FUNCTION_BLOCK SPLIT_AL_INTO_AX (* this Function splits the 64 AX (BOOL) adapters from a AL (LWORD) *)
  (* Standard: 61499-2; Description: Copyright (c) 2026 Meisterschulen am Ostbahnhof SPDX-License-Identifier: EPL-2.0 *)
  (* Version 1.0, 2026-05-16, Franz Höpfinger, Meisterschulen am Ostbahnhof, initial API and implementation and/or initial documentation *)
  PACKAGE adapter::splitting;
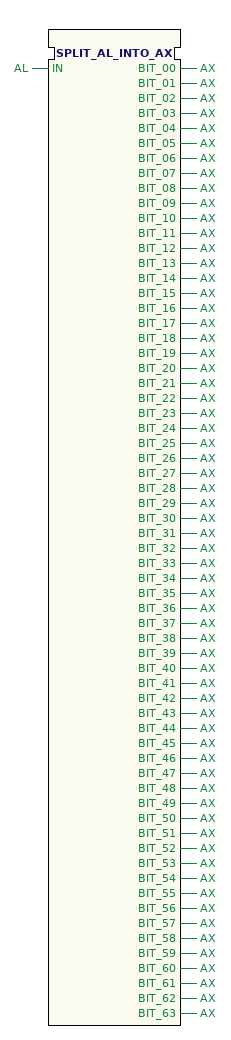
  SOCKETS
    IN : adapter::types::unidirectional::AL; (* LWORD Input *)
  END_SOCKETS
  PLUGS
    BIT_00 : adapter::types::unidirectional::AX; (* Bool Bit 0 *)
    BIT_01 : adapter::types::unidirectional::AX; (* Bool Bit 1 *)
    BIT_02 : adapter::types::unidirectional::AX; (* Bool Bit 2 *)
    BIT_03 : adapter::types::unidirectional::AX; (* Bool Bit 3 *)
    BIT_04 : adapter::types::unidirectional::AX; (* Bool Bit 4 *)
    BIT_05 : adapter::types::unidirectional::AX; (* Bool Bit 5 *)
    BIT_06 : adapter::types::unidirectional::AX; (* Bool Bit 6 *)
    BIT_07 : adapter::types::unidirectional::AX; (* Bool Bit 7 *)
    BIT_08 : adapter::types::unidirectional::AX; (* Bool Bit 8 *)
    BIT_09 : adapter::types::unidirectional::AX; (* Bool Bit 9 *)
    BIT_10 : adapter::types::unidirectional::AX; (* Bool Bit 10 *)
    BIT_11 : adapter::types::unidirectional::AX; (* Bool Bit 11 *)
    BIT_12 : adapter::types::unidirectional::AX; (* Bool Bit 12 *)
    BIT_13 : adapter::types::unidirectional::AX; (* Bool Bit 13 *)
    BIT_14 : adapter::types::unidirectional::AX; (* Bool Bit 14 *)
    BIT_15 : adapter::types::unidirectional::AX; (* Bool Bit 15 *)
    BIT_16 : adapter::types::unidirectional::AX; (* Bool Bit 16 *)
    BIT_17 : adapter::types::unidirectional::AX; (* Bool Bit 17 *)
    BIT_18 : adapter::types::unidirectional::AX; (* Bool Bit 18 *)
    BIT_19 : adapter::types::unidirectional::AX; (* Bool Bit 19 *)
    BIT_20 : adapter::types::unidirectional::AX; (* Bool Bit 20 *)
    BIT_21 : adapter::types::unidirectional::AX; (* Bool Bit 21 *)
    BIT_22 : adapter::types::unidirectional::AX; (* Bool Bit 22 *)
    BIT_23 : adapter::types::unidirectional::AX; (* Bool Bit 23 *)
    BIT_24 : adapter::types::unidirectional::AX; (* Bool Bit 24 *)
    BIT_25 : adapter::types::unidirectional::AX; (* Bool Bit 25 *)
    BIT_26 : adapter::types::unidirectional::AX; (* Bool Bit 26 *)
    BIT_27 : adapter::types::unidirectional::AX; (* Bool Bit 27 *)
    BIT_28 : adapter::types::unidirectional::AX; (* Bool Bit 28 *)
    BIT_29 : adapter::types::unidirectional::AX; (* Bool Bit 29 *)
    BIT_30 : adapter::types::unidirectional::AX; (* Bool Bit 30 *)
    BIT_31 : adapter::types::unidirectional::AX; (* Bool Bit 31 *)
    BIT_32 : adapter::types::unidirectional::AX; (* Bool Bit 32 *)
    BIT_33 : adapter::types::unidirectional::AX; (* Bool Bit 33 *)
    BIT_34 : adapter::types::unidirectional::AX; (* Bool Bit 34 *)
    BIT_35 : adapter::types::unidirectional::AX; (* Bool Bit 35 *)
    BIT_36 : adapter::types::unidirectional::AX; (* Bool Bit 36 *)
    BIT_37 : adapter::types::unidirectional::AX; (* Bool Bit 37 *)
    BIT_38 : adapter::types::unidirectional::AX; (* Bool Bit 38 *)
    BIT_39 : adapter::types::unidirectional::AX; (* Bool Bit 39 *)
    BIT_40 : adapter::types::unidirectional::AX; (* Bool Bit 40 *)
    BIT_41 : adapter::types::unidirectional::AX; (* Bool Bit 41 *)
    BIT_42 : adapter::types::unidirectional::AX; (* Bool Bit 42 *)
    BIT_43 : adapter::types::unidirectional::AX; (* Bool Bit 43 *)
    BIT_44 : adapter::types::unidirectional::AX; (* Bool Bit 44 *)
    BIT_45 : adapter::types::unidirectional::AX; (* Bool Bit 45 *)
    BIT_46 : adapter::types::unidirectional::AX; (* Bool Bit 46 *)
    BIT_47 : adapter::types::unidirectional::AX; (* Bool Bit 47 *)
    BIT_48 : adapter::types::unidirectional::AX; (* Bool Bit 48 *)
    BIT_49 : adapter::types::unidirectional::AX; (* Bool Bit 49 *)
    BIT_50 : adapter::types::unidirectional::AX; (* Bool Bit 50 *)
    BIT_51 : adapter::types::unidirectional::AX; (* Bool Bit 51 *)
    BIT_52 : adapter::types::unidirectional::AX; (* Bool Bit 52 *)
    BIT_53 : adapter::types::unidirectional::AX; (* Bool Bit 53 *)
    BIT_54 : adapter::types::unidirectional::AX; (* Bool Bit 54 *)
    BIT_55 : adapter::types::unidirectional::AX; (* Bool Bit 55 *)
    BIT_56 : adapter::types::unidirectional::AX; (* Bool Bit 56 *)
    BIT_57 : adapter::types::unidirectional::AX; (* Bool Bit 57 *)
    BIT_58 : adapter::types::unidirectional::AX; (* Bool Bit 58 *)
    BIT_59 : adapter::types::unidirectional::AX; (* Bool Bit 59 *)
    BIT_60 : adapter::types::unidirectional::AX; (* Bool Bit 60 *)
    BIT_61 : adapter::types::unidirectional::AX; (* Bool Bit 61 *)
    BIT_62 : adapter::types::unidirectional::AX; (* Bool Bit 62 *)
    BIT_63 : adapter::types::unidirectional::AX; (* Bool Bit 63 *)
  END_PLUGS
  FBS
    E_D_FF_00 : iec61499::events::E_D_FF;
    E_D_FF_01 : iec61499::events::E_D_FF;
    E_D_FF_02 : iec61499::events::E_D_FF;
    E_D_FF_03 : iec61499::events::E_D_FF;
    E_D_FF_04 : iec61499::events::E_D_FF;
    E_D_FF_05 : iec61499::events::E_D_FF;
    E_D_FF_06 : iec61499::events::E_D_FF;
    E_D_FF_07 : iec61499::events::E_D_FF;
    E_D_FF_08 : iec61499::events::E_D_FF;
    E_D_FF_09 : iec61499::events::E_D_FF;
    E_D_FF_10 : iec61499::events::E_D_FF;
    E_D_FF_11 : iec61499::events::E_D_FF;
    E_D_FF_12 : iec61499::events::E_D_FF;
    E_D_FF_13 : iec61499::events::E_D_FF;
    E_D_FF_14 : iec61499::events::E_D_FF;
    E_D_FF_15 : iec61499::events::E_D_FF;
    E_D_FF_16 : iec61499::events::E_D_FF;
    E_D_FF_17 : iec61499::events::E_D_FF;
    E_D_FF_18 : iec61499::events::E_D_FF;
    E_D_FF_19 : iec61499::events::E_D_FF;
    E_D_FF_20 : iec61499::events::E_D_FF;
    E_D_FF_21 : iec61499::events::E_D_FF;
    E_D_FF_22 : iec61499::events::E_D_FF;
    E_D_FF_23 : iec61499::events::E_D_FF;
    E_D_FF_24 : iec61499::events::E_D_FF;
    E_D_FF_25 : iec61499::events::E_D_FF;
    E_D_FF_26 : iec61499::events::E_D_FF;
    E_D_FF_27 : iec61499::events::E_D_FF;
    E_D_FF_28 : iec61499::events::E_D_FF;
    E_D_FF_29 : iec61499::events::E_D_FF;
    E_D_FF_30 : iec61499::events::E_D_FF;
    E_D_FF_31 : iec61499::events::E_D_FF;
    E_D_FF_32 : iec61499::events::E_D_FF;
    E_D_FF_33 : iec61499::events::E_D_FF;
    E_D_FF_34 : iec61499::events::E_D_FF;
    E_D_FF_35 : iec61499::events::E_D_FF;
    E_D_FF_36 : iec61499::events::E_D_FF;
    E_D_FF_37 : iec61499::events::E_D_FF;
    E_D_FF_38 : iec61499::events::E_D_FF;
    E_D_FF_39 : iec61499::events::E_D_FF;
    E_D_FF_40 : iec61499::events::E_D_FF;
    E_D_FF_41 : iec61499::events::E_D_FF;
    E_D_FF_42 : iec61499::events::E_D_FF;
    E_D_FF_43 : iec61499::events::E_D_FF;
    E_D_FF_44 : iec61499::events::E_D_FF;
    E_D_FF_45 : iec61499::events::E_D_FF;
    E_D_FF_46 : iec61499::events::E_D_FF;
    E_D_FF_47 : iec61499::events::E_D_FF;
    E_D_FF_48 : iec61499::events::E_D_FF;
    E_D_FF_49 : iec61499::events::E_D_FF;
    E_D_FF_50 : iec61499::events::E_D_FF;
    E_D_FF_51 : iec61499::events::E_D_FF;
    E_D_FF_52 : iec61499::events::E_D_FF;
    E_D_FF_53 : iec61499::events::E_D_FF;
    E_D_FF_54 : iec61499::events::E_D_FF;
    E_D_FF_55 : iec61499::events::E_D_FF;
    E_D_FF_56 : iec61499::events::E_D_FF;
    E_D_FF_57 : iec61499::events::E_D_FF;
    E_D_FF_58 : iec61499::events::E_D_FF;
    E_D_FF_59 : iec61499::events::E_D_FF;
    E_D_FF_60 : iec61499::events::E_D_FF;
    E_D_FF_61 : iec61499::events::E_D_FF;
    E_D_FF_62 : iec61499::events::E_D_FF;
    E_D_FF_63 : iec61499::events::E_D_FF;
    SPLIT_LWORD_INTO_BOOLS : eclipse4diac::utils::splitting::SPLIT_LWORD_INTO_BOOLS;
  END_FBS
  EVENT_CONNECTIONS
    IN.E1 TO SPLIT_LWORD_INTO_BOOLS.REQ;
    SPLIT_LWORD_INTO_BOOLS.CNF TO E_D_FF_00.CLK;
    SPLIT_LWORD_INTO_BOOLS.CNF TO E_D_FF_01.CLK;
    SPLIT_LWORD_INTO_BOOLS.CNF TO E_D_FF_02.CLK;
    SPLIT_LWORD_INTO_BOOLS.CNF TO E_D_FF_03.CLK;
    SPLIT_LWORD_INTO_BOOLS.CNF TO E_D_FF_04.CLK;
    SPLIT_LWORD_INTO_BOOLS.CNF TO E_D_FF_05.CLK;
    SPLIT_LWORD_INTO_BOOLS.CNF TO E_D_FF_06.CLK;
    SPLIT_LWORD_INTO_BOOLS.CNF TO E_D_FF_07.CLK;
    SPLIT_LWORD_INTO_BOOLS.CNF TO E_D_FF_08.CLK;
    SPLIT_LWORD_INTO_BOOLS.CNF TO E_D_FF_09.CLK;
    SPLIT_LWORD_INTO_BOOLS.CNF TO E_D_FF_10.CLK;
    SPLIT_LWORD_INTO_BOOLS.CNF TO E_D_FF_11.CLK;
    SPLIT_LWORD_INTO_BOOLS.CNF TO E_D_FF_12.CLK;
    SPLIT_LWORD_INTO_BOOLS.CNF TO E_D_FF_13.CLK;
    SPLIT_LWORD_INTO_BOOLS.CNF TO E_D_FF_14.CLK;
    SPLIT_LWORD_INTO_BOOLS.CNF TO E_D_FF_15.CLK;
    SPLIT_LWORD_INTO_BOOLS.CNF TO E_D_FF_16.CLK;
    SPLIT_LWORD_INTO_BOOLS.CNF TO E_D_FF_17.CLK;
    SPLIT_LWORD_INTO_BOOLS.CNF TO E_D_FF_18.CLK;
    SPLIT_LWORD_INTO_BOOLS.CNF TO E_D_FF_19.CLK;
    SPLIT_LWORD_INTO_BOOLS.CNF TO E_D_FF_20.CLK;
    SPLIT_LWORD_INTO_BOOLS.CNF TO E_D_FF_21.CLK;
    SPLIT_LWORD_INTO_BOOLS.CNF TO E_D_FF_22.CLK;
    SPLIT_LWORD_INTO_BOOLS.CNF TO E_D_FF_23.CLK;
    SPLIT_LWORD_INTO_BOOLS.CNF TO E_D_FF_24.CLK;
    SPLIT_LWORD_INTO_BOOLS.CNF TO E_D_FF_25.CLK;
    SPLIT_LWORD_INTO_BOOLS.CNF TO E_D_FF_26.CLK;
    SPLIT_LWORD_INTO_BOOLS.CNF TO E_D_FF_27.CLK;
    SPLIT_LWORD_INTO_BOOLS.CNF TO E_D_FF_28.CLK;
    SPLIT_LWORD_INTO_BOOLS.CNF TO E_D_FF_29.CLK;
    SPLIT_LWORD_INTO_BOOLS.CNF TO E_D_FF_30.CLK;
    SPLIT_LWORD_INTO_BOOLS.CNF TO E_D_FF_31.CLK;
    SPLIT_LWORD_INTO_BOOLS.CNF TO E_D_FF_32.CLK;
    SPLIT_LWORD_INTO_BOOLS.CNF TO E_D_FF_33.CLK;
    SPLIT_LWORD_INTO_BOOLS.CNF TO E_D_FF_34.CLK;
    SPLIT_LWORD_INTO_BOOLS.CNF TO E_D_FF_35.CLK;
    SPLIT_LWORD_INTO_BOOLS.CNF TO E_D_FF_36.CLK;
    SPLIT_LWORD_INTO_BOOLS.CNF TO E_D_FF_37.CLK;
    SPLIT_LWORD_INTO_BOOLS.CNF TO E_D_FF_38.CLK;
    SPLIT_LWORD_INTO_BOOLS.CNF TO E_D_FF_39.CLK;
    SPLIT_LWORD_INTO_BOOLS.CNF TO E_D_FF_40.CLK;
    SPLIT_LWORD_INTO_BOOLS.CNF TO E_D_FF_41.CLK;
    SPLIT_LWORD_INTO_BOOLS.CNF TO E_D_FF_42.CLK;
    SPLIT_LWORD_INTO_BOOLS.CNF TO E_D_FF_43.CLK;
    SPLIT_LWORD_INTO_BOOLS.CNF TO E_D_FF_44.CLK;
    SPLIT_LWORD_INTO_BOOLS.CNF TO E_D_FF_45.CLK;
    SPLIT_LWORD_INTO_BOOLS.CNF TO E_D_FF_46.CLK;
    SPLIT_LWORD_INTO_BOOLS.CNF TO E_D_FF_47.CLK;
    SPLIT_LWORD_INTO_BOOLS.CNF TO E_D_FF_48.CLK;
    SPLIT_LWORD_INTO_BOOLS.CNF TO E_D_FF_49.CLK;
    SPLIT_LWORD_INTO_BOOLS.CNF TO E_D_FF_50.CLK;
    SPLIT_LWORD_INTO_BOOLS.CNF TO E_D_FF_51.CLK;
    SPLIT_LWORD_INTO_BOOLS.CNF TO E_D_FF_52.CLK;
    SPLIT_LWORD_INTO_BOOLS.CNF TO E_D_FF_53.CLK;
    SPLIT_LWORD_INTO_BOOLS.CNF TO E_D_FF_54.CLK;
    SPLIT_LWORD_INTO_BOOLS.CNF TO E_D_FF_55.CLK;
    SPLIT_LWORD_INTO_BOOLS.CNF TO E_D_FF_56.CLK;
    SPLIT_LWORD_INTO_BOOLS.CNF TO E_D_FF_57.CLK;
    SPLIT_LWORD_INTO_BOOLS.CNF TO E_D_FF_58.CLK;
    SPLIT_LWORD_INTO_BOOLS.CNF TO E_D_FF_59.CLK;
    SPLIT_LWORD_INTO_BOOLS.CNF TO E_D_FF_60.CLK;
    SPLIT_LWORD_INTO_BOOLS.CNF TO E_D_FF_61.CLK;
    SPLIT_LWORD_INTO_BOOLS.CNF TO E_D_FF_62.CLK;
    SPLIT_LWORD_INTO_BOOLS.CNF TO E_D_FF_63.CLK;
    E_D_FF_00.EO TO BIT_00.E1;
    E_D_FF_01.EO TO BIT_01.E1;
    E_D_FF_02.EO TO BIT_02.E1;
    E_D_FF_03.EO TO BIT_03.E1;
    E_D_FF_04.EO TO BIT_04.E1;
    E_D_FF_05.EO TO BIT_05.E1;
    E_D_FF_06.EO TO BIT_06.E1;
    E_D_FF_07.EO TO BIT_07.E1;
    E_D_FF_08.EO TO BIT_08.E1;
    E_D_FF_09.EO TO BIT_09.E1;
    E_D_FF_10.EO TO BIT_10.E1;
    E_D_FF_11.EO TO BIT_11.E1;
    E_D_FF_12.EO TO BIT_12.E1;
    E_D_FF_13.EO TO BIT_13.E1;
    E_D_FF_14.EO TO BIT_14.E1;
    E_D_FF_15.EO TO BIT_15.E1;
    E_D_FF_16.EO TO BIT_16.E1;
    E_D_FF_17.EO TO BIT_17.E1;
    E_D_FF_18.EO TO BIT_18.E1;
    E_D_FF_19.EO TO BIT_19.E1;
    E_D_FF_20.EO TO BIT_20.E1;
    E_D_FF_21.EO TO BIT_21.E1;
    E_D_FF_22.EO TO BIT_22.E1;
    E_D_FF_23.EO TO BIT_23.E1;
    E_D_FF_24.EO TO BIT_24.E1;
    E_D_FF_25.EO TO BIT_25.E1;
    E_D_FF_26.EO TO BIT_26.E1;
    E_D_FF_27.EO TO BIT_27.E1;
    E_D_FF_28.EO TO BIT_28.E1;
    E_D_FF_29.EO TO BIT_29.E1;
    E_D_FF_30.EO TO BIT_30.E1;
    E_D_FF_31.EO TO BIT_31.E1;
    E_D_FF_32.EO TO BIT_32.E1;
    E_D_FF_33.EO TO BIT_33.E1;
    E_D_FF_34.EO TO BIT_34.E1;
    E_D_FF_35.EO TO BIT_35.E1;
    E_D_FF_36.EO TO BIT_36.E1;
    E_D_FF_37.EO TO BIT_37.E1;
    E_D_FF_38.EO TO BIT_38.E1;
    E_D_FF_39.EO TO BIT_39.E1;
    E_D_FF_40.EO TO BIT_40.E1;
    E_D_FF_41.EO TO BIT_41.E1;
    E_D_FF_42.EO TO BIT_42.E1;
    E_D_FF_43.EO TO BIT_43.E1;
    E_D_FF_44.EO TO BIT_44.E1;
    E_D_FF_45.EO TO BIT_45.E1;
    E_D_FF_46.EO TO BIT_46.E1;
    E_D_FF_47.EO TO BIT_47.E1;
    E_D_FF_48.EO TO BIT_48.E1;
    E_D_FF_49.EO TO BIT_49.E1;
    E_D_FF_50.EO TO BIT_50.E1;
    E_D_FF_51.EO TO BIT_51.E1;
    E_D_FF_52.EO TO BIT_52.E1;
    E_D_FF_53.EO TO BIT_53.E1;
    E_D_FF_54.EO TO BIT_54.E1;
    E_D_FF_55.EO TO BIT_55.E1;
    E_D_FF_56.EO TO BIT_56.E1;
    E_D_FF_57.EO TO BIT_57.E1;
    E_D_FF_58.EO TO BIT_58.E1;
    E_D_FF_59.EO TO BIT_59.E1;
    E_D_FF_60.EO TO BIT_60.E1;
    E_D_FF_61.EO TO BIT_61.E1;
    E_D_FF_62.EO TO BIT_62.E1;
    E_D_FF_63.EO TO BIT_63.E1;
  END_CONNECTIONS
  DATA_CONNECTIONS
    IN.D1 TO SPLIT_LWORD_INTO_BOOLS.IN;
    SPLIT_LWORD_INTO_BOOLS.BIT_63 TO E_D_FF_63.D;
    SPLIT_LWORD_INTO_BOOLS.BIT_62 TO E_D_FF_62.D;
    SPLIT_LWORD_INTO_BOOLS.BIT_61 TO E_D_FF_61.D;
    SPLIT_LWORD_INTO_BOOLS.BIT_60 TO E_D_FF_60.D;
    SPLIT_LWORD_INTO_BOOLS.BIT_59 TO E_D_FF_59.D;
    SPLIT_LWORD_INTO_BOOLS.BIT_58 TO E_D_FF_58.D;
    SPLIT_LWORD_INTO_BOOLS.BIT_57 TO E_D_FF_57.D;
    SPLIT_LWORD_INTO_BOOLS.BIT_56 TO E_D_FF_56.D;
    SPLIT_LWORD_INTO_BOOLS.BIT_55 TO E_D_FF_55.D;
    SPLIT_LWORD_INTO_BOOLS.BIT_54 TO E_D_FF_54.D;
    SPLIT_LWORD_INTO_BOOLS.BIT_53 TO E_D_FF_53.D;
    SPLIT_LWORD_INTO_BOOLS.BIT_52 TO E_D_FF_52.D;
    SPLIT_LWORD_INTO_BOOLS.BIT_51 TO E_D_FF_51.D;
    SPLIT_LWORD_INTO_BOOLS.BIT_50 TO E_D_FF_50.D;
    SPLIT_LWORD_INTO_BOOLS.BIT_49 TO E_D_FF_49.D;
    SPLIT_LWORD_INTO_BOOLS.BIT_48 TO E_D_FF_48.D;
    SPLIT_LWORD_INTO_BOOLS.BIT_47 TO E_D_FF_47.D;
    SPLIT_LWORD_INTO_BOOLS.BIT_46 TO E_D_FF_46.D;
    SPLIT_LWORD_INTO_BOOLS.BIT_45 TO E_D_FF_45.D;
    SPLIT_LWORD_INTO_BOOLS.BIT_44 TO E_D_FF_44.D;
    SPLIT_LWORD_INTO_BOOLS.BIT_43 TO E_D_FF_43.D;
    SPLIT_LWORD_INTO_BOOLS.BIT_42 TO E_D_FF_42.D;
    SPLIT_LWORD_INTO_BOOLS.BIT_41 TO E_D_FF_41.D;
    SPLIT_LWORD_INTO_BOOLS.BIT_40 TO E_D_FF_40.D;
    SPLIT_LWORD_INTO_BOOLS.BIT_39 TO E_D_FF_39.D;
    SPLIT_LWORD_INTO_BOOLS.BIT_38 TO E_D_FF_38.D;
    SPLIT_LWORD_INTO_BOOLS.BIT_37 TO E_D_FF_37.D;
    SPLIT_LWORD_INTO_BOOLS.BIT_36 TO E_D_FF_36.D;
    SPLIT_LWORD_INTO_BOOLS.BIT_35 TO E_D_FF_35.D;
    SPLIT_LWORD_INTO_BOOLS.BIT_34 TO E_D_FF_34.D;
    SPLIT_LWORD_INTO_BOOLS.BIT_33 TO E_D_FF_33.D;
    SPLIT_LWORD_INTO_BOOLS.BIT_32 TO E_D_FF_32.D;
    SPLIT_LWORD_INTO_BOOLS.BIT_31 TO E_D_FF_31.D;
    SPLIT_LWORD_INTO_BOOLS.BIT_30 TO E_D_FF_30.D;
    SPLIT_LWORD_INTO_BOOLS.BIT_29 TO E_D_FF_29.D;
    SPLIT_LWORD_INTO_BOOLS.BIT_28 TO E_D_FF_28.D;
    SPLIT_LWORD_INTO_BOOLS.BIT_27 TO E_D_FF_27.D;
    SPLIT_LWORD_INTO_BOOLS.BIT_26 TO E_D_FF_26.D;
    SPLIT_LWORD_INTO_BOOLS.BIT_25 TO E_D_FF_25.D;
    SPLIT_LWORD_INTO_BOOLS.BIT_24 TO E_D_FF_24.D;
    SPLIT_LWORD_INTO_BOOLS.BIT_23 TO E_D_FF_23.D;
    SPLIT_LWORD_INTO_BOOLS.BIT_22 TO E_D_FF_22.D;
    SPLIT_LWORD_INTO_BOOLS.BIT_21 TO E_D_FF_21.D;
    SPLIT_LWORD_INTO_BOOLS.BIT_20 TO E_D_FF_20.D;
    SPLIT_LWORD_INTO_BOOLS.BIT_19 TO E_D_FF_19.D;
    SPLIT_LWORD_INTO_BOOLS.BIT_18 TO E_D_FF_18.D;
    SPLIT_LWORD_INTO_BOOLS.BIT_17 TO E_D_FF_17.D;
    SPLIT_LWORD_INTO_BOOLS.BIT_16 TO E_D_FF_16.D;
    SPLIT_LWORD_INTO_BOOLS.BIT_15 TO E_D_FF_15.D;
    SPLIT_LWORD_INTO_BOOLS.BIT_14 TO E_D_FF_14.D;
    SPLIT_LWORD_INTO_BOOLS.BIT_13 TO E_D_FF_13.D;
    SPLIT_LWORD_INTO_BOOLS.BIT_12 TO E_D_FF_12.D;
    SPLIT_LWORD_INTO_BOOLS.BIT_11 TO E_D_FF_11.D;
    SPLIT_LWORD_INTO_BOOLS.BIT_10 TO E_D_FF_10.D;
    SPLIT_LWORD_INTO_BOOLS.BIT_09 TO E_D_FF_09.D;
    SPLIT_LWORD_INTO_BOOLS.BIT_08 TO E_D_FF_08.D;
    SPLIT_LWORD_INTO_BOOLS.BIT_07 TO E_D_FF_07.D;
    SPLIT_LWORD_INTO_BOOLS.BIT_06 TO E_D_FF_06.D;
    SPLIT_LWORD_INTO_BOOLS.BIT_05 TO E_D_FF_05.D;
    SPLIT_LWORD_INTO_BOOLS.BIT_04 TO E_D_FF_04.D;
    SPLIT_LWORD_INTO_BOOLS.BIT_03 TO E_D_FF_03.D;
    SPLIT_LWORD_INTO_BOOLS.BIT_02 TO E_D_FF_02.D;
    SPLIT_LWORD_INTO_BOOLS.BIT_01 TO E_D_FF_01.D;
    SPLIT_LWORD_INTO_BOOLS.BIT_00 TO E_D_FF_00.D;
    E_D_FF_00.Q TO BIT_00.D1;
    E_D_FF_01.Q TO BIT_01.D1;
    E_D_FF_02.Q TO BIT_02.D1;
    E_D_FF_03.Q TO BIT_03.D1;
    E_D_FF_04.Q TO BIT_04.D1;
    E_D_FF_05.Q TO BIT_05.D1;
    E_D_FF_06.Q TO BIT_06.D1;
    E_D_FF_07.Q TO BIT_07.D1;
    E_D_FF_08.Q TO BIT_08.D1;
    E_D_FF_09.Q TO BIT_09.D1;
    E_D_FF_10.Q TO BIT_10.D1;
    E_D_FF_11.Q TO BIT_11.D1;
    E_D_FF_12.Q TO BIT_12.D1;
    E_D_FF_13.Q TO BIT_13.D1;
    E_D_FF_14.Q TO BIT_14.D1;
    E_D_FF_15.Q TO BIT_15.D1;
    E_D_FF_16.Q TO BIT_16.D1;
    E_D_FF_17.Q TO BIT_17.D1;
    E_D_FF_18.Q TO BIT_18.D1;
    E_D_FF_19.Q TO BIT_19.D1;
    E_D_FF_20.Q TO BIT_20.D1;
    E_D_FF_21.Q TO BIT_21.D1;
    E_D_FF_22.Q TO BIT_22.D1;
    E_D_FF_23.Q TO BIT_23.D1;
    E_D_FF_24.Q TO BIT_24.D1;
    E_D_FF_25.Q TO BIT_25.D1;
    E_D_FF_26.Q TO BIT_26.D1;
    E_D_FF_27.Q TO BIT_27.D1;
    E_D_FF_28.Q TO BIT_28.D1;
    E_D_FF_29.Q TO BIT_29.D1;
    E_D_FF_30.Q TO BIT_30.D1;
    E_D_FF_31.Q TO BIT_31.D1;
    E_D_FF_32.Q TO BIT_32.D1;
    E_D_FF_33.Q TO BIT_33.D1;
    E_D_FF_34.Q TO BIT_34.D1;
    E_D_FF_35.Q TO BIT_35.D1;
    E_D_FF_36.Q TO BIT_36.D1;
    E_D_FF_37.Q TO BIT_37.D1;
    E_D_FF_38.Q TO BIT_38.D1;
    E_D_FF_39.Q TO BIT_39.D1;
    E_D_FF_40.Q TO BIT_40.D1;
    E_D_FF_41.Q TO BIT_41.D1;
    E_D_FF_42.Q TO BIT_42.D1;
    E_D_FF_43.Q TO BIT_43.D1;
    E_D_FF_44.Q TO BIT_44.D1;
    E_D_FF_45.Q TO BIT_45.D1;
    E_D_FF_46.Q TO BIT_46.D1;
    E_D_FF_47.Q TO BIT_47.D1;
    E_D_FF_48.Q TO BIT_48.D1;
    E_D_FF_49.Q TO BIT_49.D1;
    E_D_FF_50.Q TO BIT_50.D1;
    E_D_FF_51.Q TO BIT_51.D1;
    E_D_FF_52.Q TO BIT_52.D1;
    E_D_FF_53.Q TO BIT_53.D1;
    E_D_FF_54.Q TO BIT_54.D1;
    E_D_FF_55.Q TO BIT_55.D1;
    E_D_FF_56.Q TO BIT_56.D1;
    E_D_FF_57.Q TO BIT_57.D1;
    E_D_FF_58.Q TO BIT_58.D1;
    E_D_FF_59.Q TO BIT_59.D1;
    E_D_FF_60.Q TO BIT_60.D1;
    E_D_FF_61.Q TO BIT_61.D1;
    E_D_FF_62.Q TO BIT_62.D1;
    E_D_FF_63.Q TO BIT_63.D1;
  END_CONNECTIONS
END_FUNCTION_BLOCK
